FUNCTION_BLOCK LT_INT (* IEC 61131-3,Table 28#9 *)
  (* Standard: 61131-3 *)
  (* Version 0.1, 2006-09-15, JHC, Holobloc Inc, Converted to Template. *)
  (* Version 0.0, 2004-12-15, JHC, Rockwell Automation, Converted from SRC format. *)
  (* Compiler header: package fb.rt.plc.comp; *)
  (* Compiler classdef: (IN1 < IN2) *)
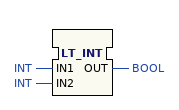
  VAR_INPUT
    IN1 : INT;
    IN2 : INT;
  END_VAR
  VAR_OUTPUT
    OUT : BOOL;
  END_VAR
END_FUNCTION_BLOCK
